FUNCTION_BLOCK FB_Conveyor
VAR_INPUT
	ins_CommIn							:Type_CommIn_Conveyor;
	inm_Reset							:BOOL;
END_VAR
VAR_OUTPUT
	outs_CommOut						:Type_CommOut_Conveyor;
	o_ProcessCycleTime					:REAL;
END_VAR
VAR
		
		m_ConveyorOn 					:BOOL;
		m_PartExists 					:BOOL;
		m_FirstCycleTime				:BOOL;
		
		int_index						:INT;
		int_index2						:INT;
		
		real_TotalCycleTime				:REAL;

		(*	Timers	*)

		T01_Init_Conveyor 				:TON;
		T02_Conveyor_On					:TON;
		T03_Piece_Found					:TON;
		T04_Conveyor_Off				:TON;
		T05_Check_Robot_Here 			:TON;
		T06_Return_Part					:TON;
				
		(*	Flags	*)
		
		SFCInit							:BOOL;
		SFCReset						:BOOL;
		SFCError						:BOOL;
		SFCPause						:BOOL;
		
		Instance_CountTotalCycleTime	:FB_CountCycleTime();
		Instance_CountProcessCycleTime	:FB_CountCycleTime();
		
		RetVal 							:enum_RetVal;
END_VAR

A01_AutomaticMode();

ACTION A01_AutomaticMode:
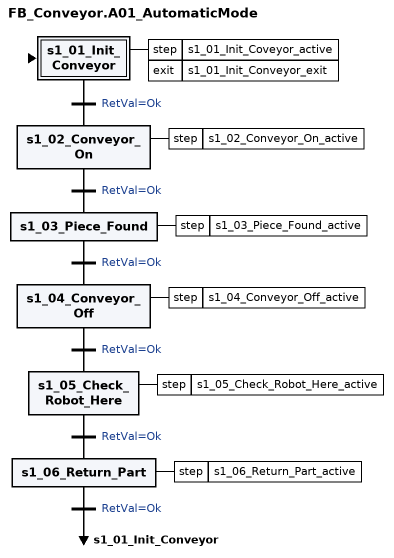
INITIAL_STEP s1_01_Init_Conveyor:
    s1_01_Init_Coveyor_active(N);  // step action
    s1_01_Init_Conveyor_exit(P0);  // exit action
END_STEP
TRANSITION FROM s1_01_Init_Conveyor TO s1_02_Conveyor_On
    := RetVal=Ok;
END_TRANSITION
STEP s1_02_Conveyor_On:  // min time T#0s, max time T#5s
    s1_02_Conveyor_On_active(N);  // step action
END_STEP
TRANSITION FROM s1_02_Conveyor_On TO s1_03_Piece_Found
    := RetVal=Ok;
END_TRANSITION
STEP s1_03_Piece_Found:
    s1_03_Piece_Found_active(N);  // step action
END_STEP
TRANSITION FROM s1_03_Piece_Found TO s1_04_Conveyor_Off
    := RetVal=Ok;
END_TRANSITION
STEP s1_04_Conveyor_Off:
    s1_04_Conveyor_Off_active(N);  // step action
END_STEP
TRANSITION FROM s1_04_Conveyor_Off TO s1_05_Check_Robot_Here
    := RetVal=Ok;
END_TRANSITION
STEP s1_05_Check_Robot_Here:
    s1_05_Check_Robot_Here_active(N);  // step action
END_STEP
TRANSITION FROM s1_05_Check_Robot_Here TO s1_06_Return_Part
    := RetVal=Ok;
END_TRANSITION
STEP s1_06_Return_Part:
    s1_06_Return_Part_active(N);  // step action
END_STEP
TRANSITION FROM s1_06_Return_Part TO s1_01_Init_Conveyor
    := RetVal=Ok;
END_TRANSITION
END_ACTION

ACTION s1_01_Init_Conveyor_exit:
IF 	NOT m_FirstCycleTime
	THEN
		o_ProcessCycleTime	:= 18;
END_IF
END_ACTION

ACTION s1_01_Init_Coveyor_active:
RetVal	:=Running;


Instance_CountTotalCycleTime(inm_TimeActive:=FALSE);

real_TotalCycleTime				:=Instance_CountTotalCycleTime.outr_CycleTime;
outs_CommOut.s_Robot.m_Ready	:=FALSE;

IF 		ins_CommIn.s_Robot.m_OutOfArea	
	THEN
		Instance_CountTotalCycleTime(inm_TimeActive:=TRUE);	
		RetVal	:=Ok;
END_IF
END_ACTION

ACTION s1_02_Conveyor_On_active:
RetVal			:=Running;
m_FirstCycleTime:=TRUE;

Instance_CountProcessCycleTime(inm_TimeActive:=TRUE);

T02_Conveyor_On(IN:=TRUE,PT:=T#15S,Q=>,ET=>);

m_ConveyorOn	:= TRUE;

IF 		T02_Conveyor_On.Q
	THEN
		T02_Conveyor_On(IN:=FALSE);
		RetVal	:=Ok;
END_IF
END_ACTION

ACTION s1_03_Piece_Found_active:
RetVal	:=Running;

T03_Piece_Found(IN:=TRUE,PT:=T#2S,Q=>,ET=>);

m_PartExists	:=TRUE; (*	Exista piesa la capatul conveyorului*)

IF 		T03_Piece_Found.Q
	THEN
		T03_Piece_Found(IN:=FALSE);
		RetVal	:=Ok;
END_IF
END_ACTION

ACTION s1_04_Conveyor_Off_active:
RetVal	:=Running;

T04_Conveyor_Off(IN:=TRUE,PT:=T#1S,Q=>,ET=>);

IF 		T04_Conveyor_Off.Q
	AND m_PartExists
	THEN
		Instance_CountProcessCycleTime(inm_TimeActive:=FALSE);
		m_PartExists:=TRUE;
		o_ProcessCycleTime			:=Instance_CountProcessCycleTime.outr_CycleTime;
		m_ConveyorOn 				:=FALSE;
		outs_CommOut.s_Robot.m_Ready:=TRUE; (* Conveyor signals Robot that the part has arrived *)
		
		T04_Conveyor_Off(IN:=FALSE);
		RetVal	:=Ok;	
END_IF
END_ACTION

ACTION s1_05_Check_Robot_Here_active:
RetVal	:=Running;
 
IF 	ins_CommIn.s_Robot.m_OutOfArea=FALSE 
	THEN 
		RetVal	:=Ok;	
END_IF
END_ACTION

ACTION s1_06_Return_Part_active:
RetVal		:=Running;
m_PartExists:=FALSE;
IF 	ins_CommIn.s_Robot.m_Work=FALSE (*	Daca robotul nu mai are treaba cu conveyorul*)
	THEN
		RetVal	:=Ok;
END_IF
END_ACTION

END_FUNCTION_BLOCK

(* stored: Version 1.1.0.1, ProductVersion 3.1.4024.3
   POU FB_Conveyor: Id {8afde770-fe0b-4e62-aad1-754bc000e997}, SpecialFunc None
   Folder S1: Id {b7c58e4a-7a97-4c8c-8d15-651110526952}
   Folder S2: Id {19a66581-18cc-4be6-846e-2238c2dfde94}
   Action A01_AutomaticMode: Id {a4f1c95d-ce24-4fd4-963a-49a535c00701}
   Action s1_01_Init_Conveyor_exit: Id {25ceec52-7a2e-47f4-bc84-0e203bee2ae4}
   Action s1_01_Init_Coveyor_active: Id {f47f3302-e853-472f-b84c-a963b1d945db}
   Action s1_02_Conveyor_On_active: Id {0bf3eaa4-d498-4982-9fe4-e8223f35d5cb}
   Action s1_03_Piece_Found_active: Id {9c850034-770e-4b64-875a-f28920c2c6b1}
   Action s1_04_Conveyor_Off_active: Id {77ebe1ee-0568-49d5-969d-d8ea8488d0a8}
   Action s1_05_Check_Robot_Here_active: Id {4cdf4ff8-d9cc-4133-b429-7d7371aba90d}
   Action s1_06_Return_Part_active: Id {bc6e2c12-a463-45d7-b6b3-738d3b4dd639} *)
